Staubli VAL3: shiftLeft.pgx

public program shiftLeft(string& x_sBinary, num x_nPos)
  local bool l_bIsBinary
  local string l_sBinary
  local num l_nIndex
begin

  l_bIsBinary=false
  call isBinary(x_sBinary, l_bIsBinary)
  l_sBinary = x_sBinary

  if l_bIsBinary
    for l_nIndex=0 to x_nPos-1
      l_sBinary = l_sBinary + "0"
    endFor
    x_sBinary=right(l_sBinary, len(x_sBinary))
  else
    logMsg("Binary->shiftLeft: wrong input format")
  endIf

end
